{attribute 'qualified_only'}
{attribute 'strict'}
TYPE eGenericInterpolatorType :
(
	XY := 1,
	XZ := 2,
	YZ := 3,
	XYZ := 4
);
END_TYPE

(* stored: Version 1.1.0.1, ProductVersion 3.1.4024.12
   DUT eGenericInterpolatorType: Id {c471b3b8-b507-48f0-b4a2-2b5de2ad876f} *)
